# B&R Automation Studio project PickAndPlace (part 2)

#### Variables.var - Local variables
```iecst
(*FB for creating a frame and reading the status of the TrackingPath*)
VAR
	MC_ReadActualPosition_Mot1 : MC_ReadActualPosition; (*FB to read the actual axis position. Used to latch the conveyor position into each created tracking frame*)
END_VAR
(*Taking Pictures*)
VAR
	CameraPV : Camera_Type := (0); (*Camera interface struct: parameters, status, input and raw detection output from the vision function*)
	ViBaseAxisBasedAcquisition_Fb : ViBaseAxisBasedAcquisition := (0); (*FB for axis-based image acquisition. Triggers images along the axis at a fixed spatial period*)
END_VAR
(*StateMachine*)
VAR CONSTANT
	MaxObjectDetectable : USINT := 8; (*Max number of objects to manage per acquisition/filtering cycle and to size arrays accordingly*)
END_VAR
VAR
	VisionState : VisionState_Enum; (*High-level vision state machine: handles readiness, acquisition, processing, frame creation, and reset*)
	Pos_mm : ARRAY[0..MaxObjectDetectable] OF Coordinate_mm_Type := [9((0))]; (*Object positions in millimeters after pixel->mm affine transform; indexed like filtered detections*)
	i : USINT := 0; (*Generic loop index for iterating detections and buffers*)
END_VAR
(**)
VAR
	UserDataSingleItemObjectRed : TrackingFrameUserDataType := (PositionType:=SingleItemPosition,SingleItemPositionData:=(PositionFilled:=TRUE,ObjectType:=Red,SyncPosUp:=(Pos:=(Z:=10+OBJECT_HEIGHT_mm)))); (*User data attached to frames for RED objects: single-item handling with Z sync offset.*)
	UserDataSingleItemObjectBlack : TrackingFrameUserDataType := (PositionType:=SingleItemPosition,SingleItemPositionData:=(PositionFilled:=TRUE,ObjectType:=Black,SyncPosUp:=(Pos:=(Z:=10+OBJECT_HEIGHT_mm)))); (*User data attached to frames for BLACK objects: single-item handling with Z sync offset.*)
	McTrkFramesDetectedObjArray : ARRAY[0..MaxObjectDetectable] OF McTrkFrmCreateParType := [9((0))]; (*Staging buffer of frames to create for all newly detected objects in the current cycle.*)
	MC_BR_DetectedObjFramesCreat : MC_BR_TrackingFramesCreate := (0); (*FB to push the staged frames (position/orientation/attributes) to the tracking path*)
END_VAR
(**)
VAR
	LastAcquisitionCount : USINT := 0; (*Memo of the last completed acquisition index to detect new images/events from the camera*)
END_VAR
(*GetTrackingPathData*)
VAR
	TrackingPathGetFramesPos_Fb : MC_BR_TrackingPathGetFrames := (0); (*FB to read existing frames on the tracking path, used to avoid creating near-duplicate frames.*)
	FramesInfo : ARRAY[0..15] OF McTrkFrmInfoType := [16((0))]; (*Buffer holding info about up to 16 existing frames fetched from the tracking path*)
	TrackingPathGetFramesPar : McTrkPathGetFrmParType := (0); (*Parameter block for the TrackingPathGetFrames FB: modes, count, and data address*)
	j : UINT := 0; (*Secondary loop index (e.g., for distance checks against existing frames or filtered objects)*)
	RedObjectFound : BOOL := FALSE; (*Flag for the current RED candidate: TRUE if not near any stored BLACK detection (valid), FALSE if too close and discarded as duplicate.*)
	CreateNewFrame : BOOL := FALSE; (*Flag deciding whether the current detection results in a new frame after distance and overlap checks*)
	Distance_px : LREAL := 0.0; (*Euclidean distance in pixels between the current suspected RED candidate and each stored BLACK detection.*)
	Distance : LREAL := 0.0; (*Computed Euclidean distance used for de-duplication/overlap checks (units: mm in frame creation step; pixels in filtering step)*)
END_VAR
VAR CONSTANT
	OBJECT_MIN_DIST : USINT := 35; (*Minimum allowed distance (mm) between a new frame and existing frames to avoid duplicates on the tracking path.*)
END_VAR
VAR
	NumbersNewFrame : USINT := 0; (*Number of frames prepared in the current cycle to be created on the tracking path. Results after the filtering*)
	CameraOutputFiltered : VF_Output_Type := (0); (*Filtered detection list combining BLACK-first and then RED objects while avoiding overlaps/doubles*)
END_VAR
(**)
VAR
	NumBlackObj : USINT := 0; (*Number of black objects detected by the camera. This value is also used when filtering red objects, since the detection models may overlap (one detects all objects, the other only black). The variable is updated at each acquisition with the current count of detected black objects.*)
END_VAR
```

#### Init.st - Init camera and getframe FB 
```iecst
ACTION CameraInitialization:
	CameraPV.Param.GainLevel := 1;
	CameraPV.Param.SetFocus := 56000;
	CameraPV.Param.ExposureTime := 2000;
	CameraPV.Param.FlashColor := 99;
	CameraPV.Param.FlashSegment := 15;
	CameraPV.Input.EnableVF := TRUE;
	CameraPV.Input.NumSearchMax := MaxObjectDetectable;
END_ACTION

ACTION GetFramesInfoInitialization:
	TrackingPathGetFramesPos_Fb.TrackingPath := ADR(gTrackingPath_1);
	TrackingPathGetFramesPar.GetMode := mcTRKPATH_GET_MOD_ALL_FRAMES;
	TrackingPathGetFramesPar.InfoMode := mcTRKPATH_INFO_MOD_ALL;
	TrackingPathGetFramesPar.NumberOfFrames := 16;
	TrackingPathGetFramesPar.DataAddress := ADR(FramesInfo);
	TrackingPathGetFramesPos_Fb.Parameters := TrackingPathGetFramesPar;
END_ACTION
```

#### FilteringOutput.st - Builds a filtered list of detections from the raw camera output
```iecst
(**
 * Derive position and color of the physical objects from the detected shapes:
 *
 * - model=2 detects only black objects, model=1 detects black and red objects
 * - Builds a filtered list of detections from the raw camera output. It first collects all BLACK objects (Model=2) into the filtered buffer.
 * - Then it evaluates each RED candidate (Model=1) and checks its Euclidean distance in pixel space against every stored BLACK object.
 * - If a RED is closer than the configured threshold (e.g., ˜100 px when using a 10000 threshold after SQRT), it is rejected to prevent counting the same physical object twice.
 * - Valid RED detections (those not overlapping a BLACK) are appended after the BLACK entries, resulting in an ordered list: BLACK first, then non-overlapping RED.
*)
ACTION CameraOutputFiltering:

	CameraOutputFiltered.NumObjFound := 0;

	FOR i := 0 TO (CameraPV.Output.NumObjFound-1)   DO

		IF CameraPV.Output.Obj[i].Model = 2 THEN
			CameraOutputFiltered.Obj[CameraOutputFiltered.NumObjFound] := CameraPV.Output.Obj[i];
			CameraOutputFiltered.NumObjFound := CameraOutputFiltered.NumObjFound + 1;
		END_IF

	END_FOR

	NumBlackObj := CameraOutputFiltered.NumObjFound;

	FOR i := 0 TO (CameraPV.Output.NumObjFound-1)   DO

		IF CameraPV.Output.Obj[i].Model = 1 THEN
			RedObjectFound := TRUE;

			IF NumBlackObj > 0 THEN

				FOR j := 0 TO NumBlackObj-1 DO
					Distance_px := SQRT(
					brmpow(LREAL_TO_REAL(CameraPV.Output.Obj[i].Pos.X - CameraOutputFiltered.Obj[j].Pos.X ), 2) +
					brmpow(LREAL_TO_REAL(CameraPV.Output.Obj[i].Pos.Y - CameraOutputFiltered.Obj[j].Pos.Y ), 2)
					);

					IF Distance_px < 10000 THEN
						RedObjectFound := FALSE;
						EXIT;
					END_IF

				END_FOR

			END_IF

			IF RedObjectFound THEN
				CameraOutputFiltered.Obj[CameraOutputFiltered.NumObjFound] := CameraPV.Output.Obj[i];
				CameraOutputFiltered.NumObjFound := CameraOutputFiltered.NumObjFound + 1;
			END_IF

		END_IF
	END_FOR

END_ACTION
```

### Program Logical/Tasks/BufferInit (IEC) - Creation of initial objects on buffer register (PLC application task)

#### Variables.var
```iecst
VAR CONSTANT
	CONV_SLOTS_MAX_IND : USINT := CONV_SLOTS-1;
	GRID : USINT := 50; (*distance between object in the register among the y direction*)
	CONV_SLOTS : USINT := 32; (*how many object can the register contain*)
	ROWS : USINT := 4; (*rows of the register*)
END_VAR
VAR
	j : USINT := 0;
	MC_BR_TrackingFrameCreate_0 : MC_BR_TrackingFramesCreate;
	TrkFrmsToCreateOnBufferRegister : ARRAY[0..CONV_SLOTS_MAX_IND] OF McTrkFrmCreateParType;
END_VAR
(*Insert your comment here.*)
VAR
	UserDataSingleItemObjectRed : TrackingFrameUserDataType := (SubFramesVisu:=[(Attribute:=RedObjectPhysicallyPresent),4(0)],PositionType:=SingleItemPosition,SingleItemPositionData:=(PositionFilled:=TRUE,ObjectType:=Red,SyncPosUp:=(Pos:=(Z:=10+OBJECT_HEIGHT_mm))));
	UserDataSingleItemObjectBlack : TrackingFrameUserDataType := (SubFramesVisu:=[(Attribute:=BlackObjectPhysicallyPresent),4(0)],PositionType:=SingleItemPosition,SingleItemPositionData:=(PositionFilled:=TRUE,ObjectType:=Black,SyncPosUp:=(Pos:=(Z:=10+OBJECT_HEIGHT_mm))));
END_VAR
```

#### Main.st
```iecst
(**
 * Buffer Initialization
 *
 * This program initializes the buffer register with a predefined grid of objects.
 * Creates tracking frames for objects positioned in a structured layout that will serve
 * as the initial inventory for the pick-and-place operations.
 *
 * Grid Layout: Objects are arranged in a rectangular grid pattern with alternating colors
 * Pattern: Red and black objects alternate (even indices = red, odd indices = black)
 * Purpose: Provides initial objects for Robot 1 to pick from buffer and place on conveyor 2
 *)

PROGRAM _INIT

	// Creation of initial objects on buffer register

	FOR j := 0 TO CONV_SLOTS_MAX_IND DO
		// X-position: Column calculation - distributes objects across columns
		TrkFrmsToCreateOnBufferRegister[j].Translation.X := GRID / 2 + GRID * (j / ROWS);
		// Y-position: Row calculation - cycles through rows (0, 1, 2, ... ROWS-1)
		TrkFrmsToCreateOnBufferRegister[j].Translation.Y := GRID / 2 + GRID * (j MOD ROWS);
		// Z-position: Object height above the buffer surface
		TrkFrmsToCreateOnBufferRegister[j].Translation.Z := OBJECT_HEIGHT_mm;

		// Alternate between red and black objects for demonstration/testing purposes
		IF (j MOD 2 = 0) THEN
			// Even indices: Red objects
			TrkFrmsToCreateOnBufferRegister[j].Attribute := HasRedObj;
			TrkFrmsToCreateOnBufferRegister[j].UserDataAddress := ADR(UserDataSingleItemObjectRed);
		ELSE
			// Odd indices: Black objects
			TrkFrmsToCreateOnBufferRegister[j].Attribute := HasBlackObj;
			TrkFrmsToCreateOnBufferRegister[j].UserDataAddress := ADR(UserDataSingleItemObjectBlack);
		END_IF;
	END_FOR;

	MC_BR_TrackingFrameCreate_0.Parameters.DataAddress := ADR(TrkFrmsToCreateOnBufferRegister);
	MC_BR_TrackingFrameCreate_0.Parameters.NumberOfFrames := CONV_SLOTS;
	MC_BR_TrackingFrameCreate_0.TrackingPath := ADR(gTrackingPath_3);

	MC_BR_TrackingFrameCreate_0.Execute := TRUE;
	MC_BR_TrackingFrameCreate_0();

END_PROGRAM

PROGRAM _EXIT
	MC_BR_TrackingFrameCreate_0();
	MC_BR_TrackingFrameCreate_0.Execute := FALSE;
END_PROGRAM
```

### Package Logical/UserPartitionData - On transfer this folder will be copied to PLC's user partition

### Package Logical/UserPartitionData/RobotMotionPrgDir - Robot programs (Motion Structured Text)

### PnpRobot1.st - Robot 1 - Single object picker (MotionST program)
```iecst
#include 'HelperFunctions.st'
#pragma LOAD 'SharedConstants.var'

(**
 * This program controls robot 1 movements and the object selection.
 * Robot 1 has a gripper for pick single products only.
 * Robot 1 has the following pick-and-place jobs to execute:
 *		1. Pick red products from conveyor belt 1 and place them to conveyor belt 2
 *		2. Pick black products from conveyor belt 1 and place them to conveyor belt 2
 *		3. Pick red products from conveyor belt 1 and place them to buffer between the conveyor belts
 *		4. Pick black products from conveyor belt 1 and place them to buffer between the conveyor belts
 *		5. Pick red products from buffer and place them to conveyor belt 2
 *		6. Pick black products from buffer and place them to conveyor belt 2
 *
 * Priority of the jobs
 *	1. Try to find an available pick-and-place sequence for job 1 or 2:
 *		1.1 Try to find a container that that will go out of workspace next and has empty positions (HasEmptyPosForRedObj|HasEmptyPosForBlackObj)
 * 			1.1.1 Try to find a pick position that can fill this container (black or red object) (HasRedObj||HasBlackObj)
 * 	2. Alternatively when no full pick-and-place sequence is available, search for a pick position only, to initiate job 3 or job 4:
 * 		2.1 First search for pick position on conveyor belt 1, when no place position is available on conveyor 2
 * 			2.1.1 Place the object to buffer (job 3 or job 4)
 * 			2.1.2 Go to waiting position with the object in the hand and wait for place positions on conveyor 2 (job 1 or job 2)
 * 	3. If no pick position available execute job 5 or job 6:
 * 		3.1 Search for products on buffer and place them on conveyor 2 (job 5 or job 6)
 *)

VAR CONSTANT
	ParkPosWithoutObject	: McPointType 	:= (Pos:=(X:=200, Y:=200, Z:= -800));
	ParkPosWithObject		: McPointType 	:= (Pos:=(X:=-200, Y:=-200, Z:= -800));
END_VAR

VAR {AT 'Mechanics'}
	MotionProgramRob1 : RobotMotionProgramType;
END_VAR

// Robot 1 helper functions

(**
 * Selects the optimal pick and place positions for the next robot operation based on priority logic.
 * Implements the job priority system: first tries complete pick-place sequences (jobs 1-2),
 * then pick-only operations to buffer (jobs 3-4), finally buffer-to-conveyor operations (jobs 5-6).
 * Automatically updates TrackingFrame UserData and Attributes for selected positions.
 *
 * @param MotionProgram: RobotMotionProgramType - IN_OUT: Motion program structure to update with selected positions
 *)
FUNCTION SelectPickPlacePositionAndSetPnpSequenceData : BOOL
	VAR_IN_OUT
		MotionProgram : RobotMotionProgramType;
	END_VAR
	VAR
		i : UINT;
	END_VAR

	// PRIORITY 1: Try to find complete pick-place sequence (jobs 1-2)
	// First, look for containers on conveyor 2 that need filling
	TrackingFrameSelectorSetAttributeMasks('Rob1_Place_Conveyor2', 0, TrackingFrameAttributeBits#HasEmptyPosForRedObj OR TrackingFrameAttributeBits#HasEmptyPosForBlackObj, 0);
	IF TrackingFrameSelect(MotionProgram.Place.TrackingFrame.ID, 'Rob1_Place_Conveyor2') THEN
		TrackingFrameGetUserData(ADR(MotionProgram.Place.TrackingFrame.UserData),
								SIZEOF(MotionProgram.Place.TrackingFrame.UserData),
								MotionProgram.Place.TrackingFrame.ID);
		// Container found on conveyor 2 - now find matching objects on conveyor 1
		FOR i := 0 TO MAX_CONTAINER_POS_INDEX DO
			IF NOT MotionProgram.Place.TrackingFrame.UserData.ContainerPositionData.ContainedPositions[i].PositionFilled THEN
				IF MotionProgram.Place.TrackingFrame.UserData.ContainerPositionData.ContainedPositions[i].ObjectType = ObjectTypeEnum#Red THEN
					// Look for red object on conveyor 1 to fill red container slot

					TrackingFrameSelectorSetAttributeMasks('Rob1_Pick_Conveyor1', 0, TrackingFrameAttributeBits#HasRedObj, 0);
					IF TrackingFrameSelect(MotionProgram.Pick.TrackingFrame.ID, 'Rob1_Pick_Conveyor1') THEN
						TrackingFrameGetUserData(ADR(MotionProgram.Pick.TrackingFrame.UserData),
												SIZEOF(MotionProgram.Pick.TrackingFrame.UserData),
												MotionProgram.Pick.TrackingFrame.ID);
						SetPickPositionBasedOnUserData(MotionProgram, TRUE, FALSE, FALSE);
						SetPlacePositionBasedOnUserData(MotionProgram, TRUE, FALSE, FALSE);
						// Complete pick-place sequence found for red object (job 1)
						EXIT; // exit for loop
					END_IF

				ELSE // Container slot expects black object
					// Look for black object on conveyor 1 to fill black container slot

					TrackingFrameSelectorSetAttributeMasks('Rob1_Pick_Conveyor1', 0, TrackingFrameAttributeBits#HasBlackObj, 0);
					IF TrackingFrameSelect(MotionProgram.Pick.TrackingFrame.ID, 'Rob1_Pick_Conveyor1') THEN
						TrackingFrameGetUserData(ADR(MotionProgram.Pick.TrackingFrame.UserData),
												SIZEOF(MotionProgram.Pick.TrackingFrame.UserData),
												MotionProgram.Pick.TrackingFrame.ID);
						SetPickPositionBasedOnUserData(MotionProgram, FALSE, TRUE, FALSE);
						SetPlacePositionBasedOnUserData(MotionProgram, FALSE, TRUE, FALSE);
						// Complete pick-place sequence found for black object (job 2)
						EXIT; // exit for loop
					END_IF
				END_IF
			END_IF
		END_FOR;

	END_IF

	// PRIORITY 2: No complete sequence found - try pick-only operations (jobs 3-4)
	IF MotionProgram.Pick.PositionSelected=FALSE THEN

		// No pick/place combination found -> Search only for pick position
		TrackingFrameSelectorSetAttributeMasks('Rob1_Pick_Conveyor1', 0, TrackingFrameAttributeBits#HasRedObj OR TrackingFrameAttributeBits#HasBlackObj, 0);
		IF TrackingFrameSelect(MotionProgram.Pick.TrackingFrame.ID, 'Rob1_Pick_Conveyor1') THEN
			TrackingFrameGetUserData(ADR(MotionProgram.Pick.TrackingFrame.UserData),
									SIZEOF(MotionProgram.Pick.TrackingFrame.UserData),
									MotionProgram.Pick.TrackingFrame.ID);
			SetPickPositionBasedOnUserData(MotionProgram, TRUE, TRUE, FALSE);
			// Robot will PickObject
		ELSE
			TrackingFrameSelectorSetAttributeMasks('Rob1_Place_Conveyor2', 0, TrackingFrameAttributeBits#HasEmptyPosForRedObj OR TrackingFrameAttributeBits#HasEmptyPosForBlackObj, 0);
			IF TrackingFrameSelect(MotionProgram.Place.TrackingFrame.ID, 'Rob1_Place_Conveyor2')  THEN
				TrackingFrameGetUserData(ADR(MotionProgram.Place.TrackingFrame.UserData),
										SIZEOF(MotionProgram.Place.TrackingFrame.UserData),
										MotionProgram.Place.TrackingFrame.ID);
				// Expected here: Container object is present on the container placeholder position
				FOR i := 0 TO MAX_CONTAINER_POS_INDEX DO
					IF NOT MotionProgram.Place.TrackingFrame.UserData.ContainerPositionData.ContainedPositions[i].PositionFilled THEN
						IF MotionProgram.Place.TrackingFrame.UserData.ContainerPositionData.ContainedPositions[i].ObjectType = ObjectTypeEnum#Red THEN

							TrackingFrameSelectorSetAttributeMasks('Rob1_PickPlace_Buffer', 0, TrackingFrameAttributeBits#HasRedObj, 0);
							IF TrackingFrameSelect(MotionProgram.Pick.TrackingFrame.ID, 'Rob1_PickPlace_Buffer') THEN
								TrackingFrameGetUserData(ADR(MotionProgram.Pick.TrackingFrame.UserData),
														SIZEOF(MotionProgram.Pick.TrackingFrame.UserData),
														MotionProgram.Pick.TrackingFrame.ID);
								SetPickPositionBasedOnUserData(MotionProgram, TRUE, FALSE, FALSE);
								SetPlacePositionBasedOnUserData(MotionProgram, TRUE, FALSE, FALSE);
								// Robot will PickObject
								EXIT; // exit for loop
							END_IF

						ELSE // TrackingFrameUserData_Place.ContainerPositionData.ContainedPositions[i].ObjectType = ObjectTypeEnum#Black
							TrackingFrameSelectorSetAttributeMasks('Rob1_PickPlace_Buffer', 0, TrackingFrameAttributeBits#HasBlackObj, 0);
							IF TrackingFrameSelect(MotionProgram.Pick.TrackingFrame.ID, 'Rob1_PickPlace_Buffer') THEN
								TrackingFrameGetUserData(ADR(MotionProgram.Pick.TrackingFrame.UserData),
														SIZEOF(MotionProgram.Pick.TrackingFrame.UserData),
														MotionProgram.Pick.TrackingFrame.ID);
								SetPickPositionBasedOnUserData(MotionProgram, FALSE, TRUE, FALSE);
								SetPlacePositionBasedOnUserData(MotionProgram, FALSE, TRUE, FALSE);
								// Robot will PickObject
								EXIT; // exit for loop
							END_IF
						END_IF
					END_IF
				END_FOR;
			END_IF
		END_IF

		// No positions selected
	END_IF
END_FUNCTION

(**
 * Selects an appropriate place position for an object that was already picked but has no place destination.
 * This function handles scenarios where the robot picked an object but couldn't immediately find a place position.
 * Prioritizes conveyor 2 containers, falls back to buffer positions if needed.
 *
 * @param MotionProgram: RobotMotionProgramType - IN_OUT: Motion program with picked object data
 *)
FUNCTION  SelectPlacePositionAndSetPlacementData : BOOL
	VAR_IN_OUT
		MotionProgram : RobotMotionProgramType;
	END_VAR
	VAR
		i : UINT;
	END_VAR

	// 1. Check type of already picked object and select place position accordingly
	IF MotionProgram.PickedObject.Type = ObjectTypeEnum#Red THEN
		TrackingFrameSelectorSetAttributeMasks('Rob1_Place_Conveyor2', 0, TrackingFrameAttributeBits#HasEmptyPosForRedObj, 0);
	ELSE // MotionProgram.PickedObject.Type = ObjectTypeEnum#Black
		TrackingFrameSelectorSetAttributeMasks('Rob1_Place_Conveyor2', 0, TrackingFrameAttributeBits#HasEmptyPosForBlackObj, 0);
	END_IF

	IF TrackingFrameSelect(MotionProgram.Place.TrackingFrame.ID, 'Rob1_Place_Conveyor2') THEN
		TrackingFrameGetUserData(ADR(MotionProgram.Place.TrackingFrame.UserData),
								SIZEOF(MotionProgram.Place.TrackingFrame.UserData),
								MotionProgram.Place.TrackingFrame.ID);
		SetPlacePositionBasedOnUserData(MotionProgram,
										MotionProgram.PickedObject.Type=ObjectTypeEnum#Red,
										MotionProgram.PickedObject.Type=ObjectTypeEnum#Black);
	ELSE
		FOR i := 0 TO MAX_CONTAINER_POS_INDEX DO
			IF MotionProgram.PickedObject.Type = ObjectTypeEnum#Red THEN
				TrackingFrameSelectorSetAttributeMasks('Rob1_PickPlace_Buffer', 0, TrackingFrameAttributeBits#HasEmptyPosForRedObj, 0);
				IF TrackingFrameSelect(MotionProgram.Place.TrackingFrame.ID, 'Rob1_PickPlace_Buffer') THEN
					TrackingFrameGetUserData(ADR(MotionProgram.Place.TrackingFrame.UserData),
											SIZEOF(MotionProgram.Place.TrackingFrame.UserData),
											MotionProgram.Place.TrackingFrame.ID);
					SetPlacePositionBasedOnUserData(MotionProgram, TRUE, FALSE);
					// Robot will PickObject
					EXIT; // exit for loop
				END_IF

			ELSE // MotionProgram.PickedObject.Type = ObjectTypeEnum#Black
				TrackingFrameSelectorSetAttributeMasks('Rob1_PickPlace_Buffer', 0, TrackingFrameAttributeBits#HasEmptyPosForBlackObj, 0);
				IF TrackingFrameSelect(MotionProgram.Place.TrackingFrame.ID, 'Rob1_PickPlace_Buffer') THEN
					TrackingFrameGetUserData(ADR(MotionProgram.Place.TrackingFrame.UserData),
											SIZEOF(MotionProgram.Place.TrackingFrame.UserData),
											MotionProgram.Place.TrackingFrame.ID);
					SetPlacePositionBasedOnUserData(MotionProgram, FALSE, TRUE);
					// Robot will PickObject
					EXIT;
				END_IF

			END_IF
		END_FOR;
	END_IF

END_FUNCTION

(**
 * Main selection function for pick and place positions when robot has no object.
 * Calls the detailed selection logic and determines the next robot state based on results.
 * Handles parking behavior when no suitable positions are found.
 *
 * @param MotionProgram: RobotMotionProgramType - IN_OUT: Motion program structure to update
 * @param FromPlacePos: BOOL - TRUE if coming from place position, FALSE if from waiting position
 *)
FUNCTION SelectPickPlacePosition : BOOL
	VAR_IN_OUT
		MotionProgram : RobotMotionProgramType;
	END_VAR
	VAR_INPUT
		FromPlacePos : BOOL; // TRUE: coming from place position, FALSE: coming from waiting position
	END_VAR

	MotionProgram.Pick.PositionSelected := FALSE;
	MotionProgram.Place.PositionSelected := FALSE;
	SelectPickPlacePositionAndSetPnpSequenceData(MotionProgram);
	IF MotionProgram.Pick.PositionSelected AND MotionProgram.Place.PositionSelected THEN
		MotionProgram.State := RobotStateEnum#PickObject;
	ELSIF MotionProgram.Pick.PositionSelected THEN
		MotionProgram.State := RobotStateEnum#PickObject;
	ELSE
		IF FromPlacePos THEN
			TrackStopR(MachineFrame, ParkPosWithoutObject, 50, 50);
			WaitEndMove();
		END_IF
		MotionProgram.State := RobotStateEnum#ParkWithNoObject;
	END_IF
END_FUNCTION

(**
 * Selects a place position for an object already held by the robot.
 * Used when robot picked an object but couldn't immediately find a place destination.
 * Handles parking behavior with object when no place position is available.
 *
 * @param MotionProgram: RobotMotionProgramType - IN_OUT: Motion program with picked object data
 * @param FromPickPos: BOOL - TRUE if coming from pick position, FALSE if from waiting position
 *)
FUNCTION SelectPlacePosition : BOOL
	VAR_IN_OUT
		MotionProgram : RobotMotionProgramType;
	END_VAR
	VAR_INPUT
		FromPickPos : BOOL; // TRUE: coming from pick position, FALSE: coming from waiting position
	END_VAR
	MotionProgram.Place.PositionSelected := FALSE;
	SelectPlacePositionAndSetPlacementData(MotionProgram);
	IF MotionProgram.Place.PositionSelected THEN
		MotionProgram.State:=RobotStateEnum#PlaceObject;
	ELSE
		IF FromPickPos THEN
			TrackStopR(MachineFrame, ParkPosWithObject, 50, 50);
			WaitEndMove();
		END_IF
		MotionProgram.State := RobotStateEnum#ParkWithGrippedObject;
	END_IF

END_FUNCTION

(**
 * Updates the products in the gripper to be shown in Scene Viewer
 *)
FUNCTION UpdateGripperContent : BOOL
	VAR_IN_OUT
		MotionProgram : RobotMotionProgramType;
	END_VAR
	VAR_INPUT
		Pick : BOOL; // TRUE: Pick operation, FALSE: Place operation
	END_VAR
	IF Pick THEN
		MotionProgram.GripperContent.RedObjectInGripper[0] := MotionProgram.PickedObject.Type = ObjectTypeEnum#Red;
		MotionProgram.GripperContent.BlackObjectInGripper[0] := MotionProgram.PickedObject.Type = ObjectTypeEnum#Black;
	ELSE
		MotionProgram.GripperContent.RedObjectInGripper[0] := FALSE;
		MotionProgram.GripperContent.BlackObjectInGripper[0] := FALSE;
	END_IF
END_FUNCTION

// Robot 1 Main Motion Program - State Machine Implementation

PROGRAM _MAIN

	MotionProgramRob1.State := RobotStateEnum#Start;

	REPEAT
		CASE MotionProgramRob1.State OF

			RobotStateEnum#Start:
				// Initialize robot to park position without object
				MoveLR(ParkPosWithoutObject);
				WaitALAP();
				MotionProgramRob1.State := RobotStateEnum#ParkWithNoObject;

			RobotStateEnum#PickObject:
				// Execute pick operation
				TrackObjectR(MotionProgramRob1.Pick.TrackingFrame.ID, MotionProgramRob1.Pick.SynchPosUp, 50, 50);
				DO_PATH_SYNCH
					MotionProgramRob1.CloseGripper := TRUE;	 // To increase throughput (reduce required WaitTime), also signaling feature could be used for activating the vaccuum
				END_PATH_SYNCH
				MoveLR(MotionProgramRob1.Pick.SynchPosDown);
				DO_PATH_SYNCH
					UpdateGripperContent(MotionProgramRob1, TRUE);
				END_PATH_SYNCH
				WaitTime(0.2);
				MoveLR(MotionProgramRob1.Pick.SynchPosUp);
				IF MotionProgramRob1.Place.PositionSelected THEN
					MotionProgramRob1.State := RobotStateEnum#PlaceObject;
				ELSE
					WaitALAP();
					SelectPlacePosition(MotionProgramRob1, TRUE);
				END_IF

			RobotStateEnum#PlaceObject:
				// Execute place operation
				TrackObjectR(MotionProgramRob1.Place.TrackingFrame.ID, MotionProgramRob1.Place.SynchPosUp, 50, 50);
				MoveLR(MotionProgramRob1.Place.SynchPosDown);
				DO_PATH_SYNCH
					MotionProgramRob1.CloseGripper := FALSE;	 // To increase throughput (reduce required WaitTime), also signaling feature could be used for deactivating the vaccuum
					UpdateGripperContent(MotionProgramRob1, FALSE);
				END_PATH_SYNCH
				WaitTime(0.1);
				MoveLR(MotionProgramRob1.Place.SynchPosUp);
				WaitALAP();
				// Look for next pick-place sequence after successful placement
				SelectPickPlacePosition(MotionProgramRob1, TRUE);

			RobotStateEnum#ParkWithNoObject:
				// Robot is parked without object - continuously search for work
				SelectPickPlacePosition(MotionProgramRob1, FALSE);

			RobotStateEnum#ParkWithGrippedObject:
				// Robot has object but no place position - search for place destination
				SelectPlacePosition(MotionProgramRob1, FALSE);

		END_CASE
	UNTIL FALSE END_REPEAT;

END_PROGRAM
```

### PnpRobot2.st - Robot 2 - Container picker (MotionST program)
```iecst
#include 'HelperFunctions.st'
#pragma LOAD 'SharedConstants.var'

(**
 * This program controls robot 2 movements and object selection.
 * Robot 2 has a gripper designed for picking entire containers (4 objects at once).
 * Robot 2 has a single pick-and-place job to execute:
 *		Pick complete containers that have been filled by robot 1 from conveyor belt 2
 *		and place them on conveyor belt 1.
 *
 * Operation: Robot 2 waits for containers on conveyor 2 that contain objects (filled by Robot 1),
 * then transfers these complete containers to conveyor 1.
 *)

VAR CONSTANT
	ParkPosWithoutObject      : McPointType := (Pos:=(X:=-200, Y:=-200, Z:= -800));
	ParkPosWithObject      : McPointType := (Pos:=(X:=200, Y:=200, Z:= -800));
END_VAR
VAR {AT 'Mechanics'}
	MotionProgramRob2 : RobotMotionProgramType;
END_VAR

// Robot 2 helper functions

(**
 * Selects a filled container on conveyor 2 for picking operation.
 * Searches for containers that contain objects (filled by Robot 1) and are ready for transfer.
 * Automatically updates TrackingFrame UserData and Attributes for the selected position.
 *
 * @param MotionProgram: RobotMotionProgramType - IN_OUT: Motion program structure to update with pick position
 *)
FUNCTION SelectPickPositionAndSetPickData : BOOL
	VAR_IN_OUT
		MotionProgram : RobotMotionProgramType;
	END_VAR
	VAR
		i : UINT;
	END_VAR

	// Search for containers on conveyor 2 that contain objects (red or black)
	TrackingFrameSelectorSetAttributeMasks('Rob2_Pick_Conveyor2', 0, TrackingFrameAttributeBits#HasRedObj OR TrackingFrameAttributeBits#HasBlackObj, 0);

	IF TrackingFrameSelect(MotionProgram.Pick.TrackingFrame.ID, 'Rob2_Pick_Conveyor2') THEN
		TrackingFrameGetUserData(ADR(MotionProgram.Pick.TrackingFrame.UserData),
								SIZEOF(MotionProgram.Pick.TrackingFrame.UserData),
								MotionProgram.Pick.TrackingFrame.ID);
		SetPickPositionBasedOnUserData(MotionProgram, FALSE, FALSE, TRUE);
		// Container selected for pickup
	END_IF
END_FUNCTION

(**
 * Selects an empty container position on conveyor 1 for placing the picked container.
 * Searches for available container placeholder positions on the destination conveyor.
 * Automatically updates TrackingFrame UserData and Attributes for the selected position.
 *
 * @param MotionProgram: RobotMotionProgramType - IN_OUT: Motion program structure to update with place position
 *)
FUNCTION  SelectPlacePositionAndSetPlacementData : BOOL
	VAR_IN_OUT
		MotionProgram : RobotMotionProgramType;
	END_VAR
	VAR
		i : UINT;
	END_VAR

	// Search for empty container positions on conveyor 1
	TrackingFrameSelectorSetAttributeMasks('Rob2_Place_Conveyor1', 0, TrackingFrameAttributeBits#HasEmptyPosForContainer, 0);
	IF TrackingFrameSelect(MotionProgram.Place.TrackingFrame.ID, 'Rob2_Place_Conveyor1') THEN
		TrackingFrameGetUserData(ADR(MotionProgram.Place.TrackingFrame.UserData),
								SIZEOF(MotionProgram.Place.TrackingFrame.UserData),
								MotionProgram.Place.TrackingFrame.ID);
		SetPlacePositionBasedOnUserData(MotionProgram, FALSE, FALSE, TRUE);
	END_IF
END_FUNCTION

(**
 * Main selection function for pick positions when robot has no container.
 * Calls the detailed pick selection logic and determines the next robot state based on results.
 * Handles parking behavior when no suitable containers are available for pickup.
 *
 * @param MotionProgram: RobotMotionProgramType - IN_OUT: Motion program structure to update
 * @param FromPlacePos: BOOL - TRUE if coming from place position, FALSE if from waiting position
 *)
FUNCTION SelectPickPosition : BOOL
	VAR_IN_OUT
		MotionProgram : RobotMotionProgramType;
	END_VAR
	VAR_INPUT
		FromPlacePos : BOOL; // TRUE: coming from place position, FALSE: coming from waiting position
	END_VAR
	MotionProgram.Pick.PositionSelected := FALSE;
	SelectPickPositionAndSetPickData(MotionProgram);
	IF MotionProgram.Pick.PositionSelected THEN
		MotionProgram.State := RobotStateEnum#PickObject;
	ELSE
		IF FromPlacePos THEN
			TrackStopR(MachineFrame, ParkPosWithoutObject, 50, 50);
			WaitEndMove();
		END_IF
		MotionProgram.State := RobotStateEnum#ParkWithNoObject;
	END_IF

END_FUNCTION

(**
 * Selects a place position for a container already held by the robot.
 * Used when robot picked a container but couldn't immediately find a place destination.
 * Handles parking behavior with container when no place position is available.
 *
 * @param MotionProgram: RobotMotionProgramType - IN_OUT: Motion program with picked container data
 * @param FromPickPos: BOOL - TRUE if coming from pick position, FALSE if from waiting position
 *)
FUNCTION SelectPlacePosition : BOOL
	VAR_IN_OUT
		MotionProgram : RobotMotionProgramType;
	END_VAR
	VAR_INPUT
		FromPickPos : BOOL; // TRUE: coming from pick position, FALSE: coming from waiting position
	END_VAR
	MotionProgram.Place.PositionSelected := FALSE;
	SelectPlacePositionAndSetPlacementData(MotionProgram);
	IF MotionProgram.Place.PositionSelected THEN
		MotionProgram.State:=RobotStateEnum#PlaceObject;
	ELSE
		IF FromPickPos THEN
			TrackStopR(MachineFrame, ParkPosWithObject, 50, 50);
			WaitEndMove();
		END_IF
		MotionProgram.State:=RobotStateEnum#ParkWithGrippedObject;
	END_IF
END_FUNCTION

(**
 *  * Updates the products in the gripper to be shown in Scene Viewer
 *)
FUNCTION UpdateGripperContent : BOOL
	VAR_IN_OUT
		MotionProgram : RobotMotionProgramType;
	END_VAR
	VAR_INPUT
		Pick : BOOL; // TRUE: Pick operation, FALSE: Place operation
	END_VAR
	IF Pick THEN
		MotionProgram.GripperContent.RedObjectInGripper[0] := MotionProgram.Pick.TrackingFrame.UserData.ContainerPositionData.ContainedPositions[0].PositionFilled AND MotionProgram.Pick.TrackingFrame.UserData.ContainerPositionData.ContainedPositions[0].ObjectType = ObjectTypeEnum#Red;
		MotionProgram.GripperContent.RedObjectInGripper[1] := MotionProgram.Pick.TrackingFrame.UserData.ContainerPositionData.ContainedPositions[1].PositionFilled AND MotionProgram.Pick.TrackingFrame.UserData.ContainerPositionData.ContainedPositions[1].ObjectType = ObjectTypeEnum#Red;
		MotionProgram.GripperContent.RedObjectInGripper[2] := MotionProgram.Pick.TrackingFrame.UserData.ContainerPositionData.ContainedPositions[2].PositionFilled AND MotionProgram.Pick.TrackingFrame.UserData.ContainerPositionData.ContainedPositions[2].ObjectType = ObjectTypeEnum#Red;
		MotionProgram.GripperContent.RedObjectInGripper[3] := MotionProgram.Pick.TrackingFrame.UserData.ContainerPositionData.ContainedPositions[3].PositionFilled AND MotionProgram.Pick.TrackingFrame.UserData.ContainerPositionData.ContainedPositions[3].ObjectType = ObjectTypeEnum#Red;

		MotionProgram.GripperContent.BlackObjectInGripper[0] := MotionProgram.Pick.TrackingFrame.UserData.ContainerPositionData.ContainedPositions[0].PositionFilled AND MotionProgram.Pick.TrackingFrame.UserData.ContainerPositionData.ContainedPositions[0].ObjectType = ObjectTypeEnum#Black;
		MotionProgram.GripperContent.BlackObjectInGripper[1] := MotionProgram.Pick.TrackingFrame.UserData.ContainerPositionData.ContainedPositions[1].PositionFilled AND MotionProgram.Pick.TrackingFrame.UserData.ContainerPositionData.ContainedPositions[1].ObjectType = ObjectTypeEnum#Black;
		MotionProgram.GripperContent.BlackObjectInGripper[2] := MotionProgram.Pick.TrackingFrame.UserData.ContainerPositionData.ContainedPositions[2].PositionFilled AND MotionProgram.Pick.TrackingFrame.UserData.ContainerPositionData.ContainedPositions[2].ObjectType = ObjectTypeEnum#Black;
		MotionProgram.GripperContent.BlackObjectInGripper[3] := MotionProgram.Pick.TrackingFrame.UserData.ContainerPositionData.ContainedPositions[3].PositionFilled AND MotionProgram.Pick.TrackingFrame.UserData.ContainerPositionData.ContainedPositions[3].ObjectType = ObjectTypeEnum#Black;
	ELSE
		MotionProgram.GripperContent.RedObjectInGripper[0] := FALSE;
		MotionProgram.GripperContent.RedObjectInGripper[1] := FALSE;
		MotionProgram.GripperContent.RedObjectInGripper[2] := FALSE;
		MotionProgram.GripperContent.RedObjectInGripper[3] := FALSE;

		MotionProgram.GripperContent.BlackObjectInGripper[0] := FALSE;
		MotionProgram.GripperContent.BlackObjectInGripper[1] := FALSE;
		MotionProgram.GripperContent.BlackObjectInGripper[2] := FALSE;
		MotionProgram.GripperContent.BlackObjectInGripper[3] := FALSE;
	END_IF
END_FUNCTION

// Robot 2 Main Motion Program - Container Transfer State Machine

PROGRAM _MAIN

	MotionProgramRob2.State := RobotStateEnum#Start;

	REPEAT
		CASE MotionProgramRob2.State OF

			RobotStateEnum#Start:
				// Initialize robot to park position
				MoveLR(ParkPosWithoutObject);
				WaitALAP();
				MotionProgramRob2.State := RobotStateEnum#ParkWithNoObject;

			RobotStateEnum#PickObject:
				// Execute container pick operation
				TrackObjectR(MotionProgramRob2.Pick.TrackingFrame.ID, MotionProgramRob2.Pick.SynchPosUp, 50, 50);
				DO_PATH_SYNCH
					MotionProgramRob2.CloseGripper := TRUE;	 // To increase throughput (reduce required WaitTime), also signaling feature could be used for deactivating the vaccuum
				END_PATH_SYNCH
				MoveLR(MotionProgramRob2.Pick.SynchPosDown);
				DO_PATH_SYNCH
					UpdateGripperContent(MotionProgramRob2, TRUE);
				END_PATH_SYNCH
				WaitTime(0.1); // Allow time for container to settle in gripper
				MoveLR(MotionProgramRob2.Pick.SynchPosUp);
				WaitALAP();
				// Search for place position after successful container pickup
				SelectPlacePosition(MotionProgramRob2, TRUE);

			RobotStateEnum#PlaceObject:
				// Execute container place operation
				TrackObjectR(MotionProgramRob2.Place.TrackingFrame.ID, MotionProgramRob2.Place.SynchPosUp, 50, 50);
				MoveLR(MotionProgramRob2.Place.SynchPosDown);
				DO_PATH_SYNCH
					MotionProgramRob2.CloseGripper := FALSE;	 // To increase throughput (reduce required WaitTime), also signaling feature could be used for deactivating the vaccuum
					UpdateGripperContent(MotionProgramRob2, FALSE);
				END_PATH_SYNCH
				WaitTime(0.05); // Brief wait for container release
				MoveLR(MotionProgramRob2.Place.SynchPosUp);
				WaitALAP();
				// Look for next container to transfer after successful placement
				SelectPickPosition(MotionProgramRob2, TRUE);

			RobotStateEnum#ParkWithNoObject:
				// Robot is parked without container - continuously search for containers to transfer
				SelectPickPosition(MotionProgramRob2, FALSE);

			RobotStateEnum#ParkWithGrippedObject:
				// Robot has container but no place position - search for place destination
				SelectPlacePosition(MotionProgramRob2, FALSE);

		END_CASE
	UNTIL FALSE END_REPEAT;

END_PROGRAM
```

### HelperFunctions.st - Helper functions for objects selection shared by both robots (MotionST functions)
```iecst
#include 'SharedTypes.typ'
#pragma LOAD 'SharedConstants.var'

(*
 * Generates and returns an attribute value (bitmask) that represents the state of the TrackingFrame userData.
 * This function analyzes the position type and object states to create appropriate attribute flags.
 *
 * @param userData: TrackingFrameUserDataType - The user data structure containing position and object information
 * @return UDINT - Bitmask representing the current state (empty positions, object types, etc.)
 *)
FUNCTION GetAttributeBasedOnUserData : UDINT
	VAR_INPUT
		userData : TrackingFrameUserDataType;
	END_VAR
	VAR
		attribute : UDINT;
		i : UINT;
	END_VAR
	attribute := 0;
	IF userData.PositionType = TrackingFramePositionTypeEnum#SingleItemPosition THEN
		IF userData.SingleItemPositionData.PositionFilled = FALSE THEN
			IF userData.SingleItemPositionData.ObjectType = ObjectTypeEnum#Red THEN
				attribute := attribute OR TrackingFrameAttributeBits#HasEmptyPosForRedObj;
			ELSE // userData.SingleItemPositionData.ObjectType = ObjectTypeEnum#Black
				attribute := attribute OR TrackingFrameAttributeBits#HasEmptyPosForBlackObj;
			END_IF
		ELSE // userData.SingleItemPositionData.PositionFilled = TRUE
			IF userData.SingleItemPositionData.ObjectType = ObjectTypeEnum#Red THEN
				attribute := attribute OR TrackingFrameAttributeBits#HasRedObj;
			ELSE // userData.SingleItemPositionData.ObjectType = ObjectTypeEnum#Black
				attribute := attribute OR TrackingFrameAttributeBits#HasBlackObj;
			END_IF
		END_IF
	ELSIF userData.PositionType = TrackingFramePositionTypeEnum#ContainerPosition THEN
		IF userData.ContainerPositionData.PositionFilled = FALSE THEN
			attribute := attribute OR TrackingFrameAttributeBits#HasEmptyPosForContainer;
		ELSE //userData.ContainerPositionData.PositionFilled = TRUE
			FOR i := 0 TO MAX_CONTAINER_POS_INDEX DO
				IF userData.ContainerPositionData.ContainedPositions[i].PositionFilled THEN
					IF userData.ContainerPositionData.ContainedPositions[i].ObjectType = ObjectTypeEnum#Red THEN
						attribute := attribute OR TrackingFrameAttributeBits#HasRedObj;
					ELSE // userData.ContainerPositionData.ContainedPositions[i].ObjectType = ObjectTypeEnum#Black
						attribute := attribute OR TrackingFrameAttributeBits#HasBlackObj;
					END_IF
				ELSE // userData.ContainerPositionData.ContainedPositions[i].PositionFilled = FALSE
					IF userData.ContainerPositionData.ContainedPositions[i].ObjectType = ObjectTypeEnum#Red THEN
						attribute := attribute OR TrackingFrameAttributeBits#HasEmptyPosForRedObj;
					ELSE // userData.ContainerPositionData.ContainedPositions[i].ObjectType = ObjectTypeEnum#Black
						attribute := attribute OR TrackingFrameAttributeBits#HasEmptyPosForBlackObj;
					END_IF
				END_IF
			END_FOR;
		END_IF
	END_IF
	GetAttributeBasedOnUserData := attribute;
END_FUNCTION

(*
 * Generates an attribute value (bitmask) and writes it directly to the specified TrackingFrame.
 * This is a convenience function that combines GetAttributeBasedOnUserData with TrackingFrameSetAttribute.
 *
 * @param trackingFrameId: McTrkFrmIdentType - The ID of the tracking frame to update
 * @param userData: TrackingFrameUserDataType - The user data to analyze for attribute generation
 * @return UDINT - The generated attribute bitmask that was written to the tracking frame
 *)
FUNCTION SetAttributeBasedOnUserData : UDINT
	VAR_INPUT
		trackingFrameId : McTrkFrmIdentType;
		userData : TrackingFrameUserDataType;
	END_VAR
	VAR
		attribute : UDINT;
	END_VAR
	attribute := GetAttributeBasedOnUserData(userData);
	TrackingFrameSetAttribute(trackingFrameId, attribute);
	SetAttributeBasedOnUserData := attribute;
END_FUNCTION

(*
 * Configures the pick operation in the MotionProgram based on selected TrackingFrame userData.
 * Updates synchronization positions, object type information, and marks the position as empty after picking.
 *
 * @param MotionProgram: RobotMotionProgramType - IN_OUT: Motion program structure to update
 * @param objectTypeRed: BOOL - TRUE if red objects should be considered for picking
 * @param objectTypeBlack: BOOL - TRUE if black objects should be considered for picking
 * @param objectTypeContainer: BOOL - TRUE to pick entire container, FALSE to pick individual contained item
 * @return BOOL - Success status of the operation
 *)
FUNCTION SetPickPositionBasedOnUserData : BOOL
	VAR_IN_OUT
		MotionProgram : RobotMotionProgramType;
	END_VAR
	VAR_INPUT
		objectTypeRed : BOOL;
		objectTypeBlack : BOOL;
		objectTypeContainer : BOOL; // TRUE the entire container will be picked, FALSE only a contained item will be picked
	END_VAR
	VAR
		i : UINT;
	END_VAR
	IF MotionProgram.Pick.TrackingFrame.UserData.PositionType = TrackingFramePositionTypeEnum#SingleItemPosition THEN
		MotionProgram.Pick.SynchPosUp := MotionProgram.Pick.TrackingFrame.UserData.SingleItemPositionData.SyncPosUp;
		MotionProgram.Pick.SynchPosDown := MotionProgram.Pick.TrackingFrame.UserData.SingleItemPositionData.SyncPosDown;
		MotionProgram.PickedObject.Type := MotionProgram.Pick.TrackingFrame.UserData.SingleItemPositionData.ObjectType;
		MotionProgram.PickedObject.ContainerIndex := 0; // No container index for single item position
		MotionProgram.Pick.TrackingFrame.UserData.SingleItemPositionData.PositionFilled := FALSE;
		MotionProgram.Pick.TrackingFrame.UserData.SubFramesVisu[0].Attribute := MotionProgram.Pick.TrackingFrame.UserData.SubFramesVisu[0].Attribute OR TrackingFrameAttributeBits#ProductSelectedForOperation;
	ELSE // MotionProgram.Pick.TrackingFrame.UserData.PositionType = TrackingFramePositionTypeEnum#ContainerPosition
		IF objectTypeContainer THEN // Entire container will be picked
			MotionProgram.Pick.SynchPosUp := MotionProgram.Pick.TrackingFrame.UserData.ContainerPositionData.SyncPosUp;
			MotionProgram.Pick.SynchPosDown := MotionProgram.Pick.TrackingFrame.UserData.ContainerPositionData.SyncPosDown;
			MotionProgram.Pick.TrackingFrame.UserData.ContainerPositionData.PositionFilled := FALSE;
			MotionProgram.Pick.TrackingFrame.UserData.SubFramesVisu[0].Attribute := MotionProgram.Pick.TrackingFrame.UserData.SubFramesVisu[0].Attribute OR TrackingFrameAttributeBits#ContainerSelectedForOperation;
		ELSE // Only a contained item will be picked
			// Search through container positions to find the requested object type
			FOR i := 0 TO MAX_CONTAINER_POS_INDEX DO
				IF MotionProgram.Pick.TrackingFrame.UserData.ContainerPositionData.ContainedPositions[i].PositionFilled THEN
					IF objectTypeRed AND MotionProgram.Pick.TrackingFrame.UserData.ContainerPositionData.ContainedPositions[i].ObjectType = ObjectTypeEnum#Red THEN
						MotionProgram.Pick.SynchPosUp := MotionProgram.Pick.TrackingFrame.UserData.ContainerPositionData.ContainedPositions[i].SyncPosUp;
						MotionProgram.Pick.SynchPosDown := MotionProgram.Pick.TrackingFrame.UserData.ContainerPositionData.ContainedPositions[i].SyncPosDown;
						MotionProgram.PickedObject.Type := MotionProgram.Pick.TrackingFrame.UserData.ContainerPositionData.ContainedPositions[i].ObjectType;
						MotionProgram.PickedObject.ContainerIndex := i;
						MotionProgram.Pick.TrackingFrame.UserData.ContainerPositionData.ContainedPositions[i].PositionFilled := FALSE;
						MotionProgram.Pick.TrackingFrame.UserData.SubFramesVisu[i+1].Attribute := MotionProgram.Pick.TrackingFrame.UserData.SubFramesVisu[i+1].Attribute OR TrackingFrameAttributeBits#ProductSelectedForOperation;
						EXIT; // exit for loop
					ELSIF objectTypeBlack AND MotionProgram.Pick.TrackingFrame.UserData.ContainerPositionData.ContainedPositions[i].ObjectType = ObjectTypeEnum#Black THEN
						MotionProgram.Pick.SynchPosUp := MotionProgram.Pick.TrackingFrame.UserData.ContainerPositionData.ContainedPositions[i].SyncPosUp;
						MotionProgram.Pick.SynchPosDown := MotionProgram.Pick.TrackingFrame.UserData.ContainerPositionData.ContainedPositions[i].SyncPosDown;
						MotionProgram.PickedObject.Type := MotionProgram.Pick.TrackingFrame.UserData.ContainerPositionData.ContainedPositions[i].ObjectType;
						MotionProgram.PickedObject.ContainerIndex := i;
						MotionProgram.Pick.TrackingFrame.UserData.ContainerPositionData.ContainedPositions[i].PositionFilled := FALSE;
						MotionProgram.Pick.TrackingFrame.UserData.SubFramesVisu[i+1].Attribute := MotionProgram.Pick.TrackingFrame.UserData.SubFramesVisu[i+1].Attribute OR TrackingFrameAttributeBits#ProductSelectedForOperation;
						EXIT; // exit for loop
					END_IF
				END_IF
			END_FOR;

		END_IF
	END_IF
	MotionProgram.Pick.PositionSelected := TRUE;
	TrackingFrameSetUserData(ADR(MotionProgram.Pick.TrackingFrame.UserData),
							SIZEOF(MotionProgram.Pick.TrackingFrame.UserData),
							MotionProgram.Pick.TrackingFrame.ID);
	MotionProgram.Pick.TrackingFrame.Attribute := SetAttributeBasedOnUserData(MotionProgram.Pick.TrackingFrame.ID, MotionProgram.Pick.TrackingFrame.UserData);
END_FUNCTION

(*
 * Configures the place operation in the MotionProgram based on selected TrackingFrame userData.
 * Updates synchronization positions, transfers object data from pick to place position, and marks position as filled.
 *
 * @param MotionProgram: RobotMotionProgramType - IN_OUT: Motion program structure to update
 * @param objectTypeRed: BOOL - TRUE if red objects should be considered for placement
 * @param objectTypeBlack: BOOL - TRUE if black objects should be considered for placement
 * @param objectTypeContainer: BOOL - TRUE to place entire container, FALSE to place individual item in container
 * @return BOOL - Success status of the operation
 *)
FUNCTION SetPlacePositionBasedOnUserData : BOOL
	VAR_IN_OUT
		MotionProgram : RobotMotionProgramType;
	END_VAR
	VAR_INPUT
		objectTypeRed : BOOL;
		objectTypeBlack : BOOL;
		objectTypeContainer : BOOL; // TRUE the entire container will be picked, FALSE only a contained item will be picked
	END_VAR
	VAR
		i : UINT;
	END_VAR
	IF MotionProgram.Place.TrackingFrame.UserData.PositionType = TrackingFramePositionTypeEnum#SingleItemPosition THEN
		MotionProgram.Place.SynchPosUp := MotionProgram.Place.TrackingFrame.UserData.SingleItemPositionData.SyncPosUp;
		MotionProgram.Place.SynchPosDown := MotionProgram.Place.TrackingFrame.UserData.SingleItemPositionData.SyncPosDown;
		// Transfer product identification from pick to place position for traceability
		MotionProgram.Place.TrackingFrame.UserData.SingleItemPositionData.ProductID := MotionProgram.Pick.TrackingFrame.UserData.SingleItemPositionData.ProductID;
		MotionProgram.Place.TrackingFrame.UserData.SingleItemPositionData.PositionFilled := TRUE;
		MotionProgram.Place.TrackingFrame.UserData.SubFramesVisu[0].Attribute := MotionProgram.Place.TrackingFrame.UserData.SubFramesVisu[0].Attribute OR TrackingFrameAttributeBits#ProductSelectedForOperation;
	ELSE // MotionProgram.Place.TrackingFrame.UserData.PositionType = TrackingFramePositionTypeEnum#ContainerPosition
		IF objectTypeContainer THEN // Entire container will be placed
			MotionProgram.Place.SynchPosUp := MotionProgram.Place.TrackingFrame.UserData.ContainerPositionData.SyncPosUp;
			MotionProgram.Place.SynchPosDown := MotionProgram.Place.TrackingFrame.UserData.ContainerPositionData.SyncPosDown;
			MotionProgram.Place.TrackingFrame.UserData.ContainerPositionData := MotionProgram.Pick.TrackingFrame.UserData.ContainerPositionData; // Copy container data from pick to place position
			MotionProgram.Place.TrackingFrame.UserData.ContainerPositionData.PositionFilled := TRUE;
			MotionProgram.Place.TrackingFrame.UserData.SubFramesVisu[0].Attribute := MotionProgram.Place.TrackingFrame.UserData.SubFramesVisu[0].Attribute OR TrackingFrameAttributeBits#ContainerSelectedForOperation;
		ELSE // Will be placed in a contained position only
			// Search for position with object present
			FOR i := 0 TO MAX_CONTAINER_POS_INDEX DO
				IF NOT MotionProgram.Place.TrackingFrame.UserData.ContainerPositionData.ContainedPositions[i].PositionFilled THEN
					IF objectTypeRed AND MotionProgram.Place.TrackingFrame.UserData.ContainerPositionData.ContainedPositions[i].ObjectType = ObjectTypeEnum#Red THEN
						MotionProgram.Place.SynchPosUp := MotionProgram.Place.TrackingFrame.UserData.ContainerPositionData.ContainedPositions[i].SyncPosUp;
						MotionProgram.Place.SynchPosDown := MotionProgram.Place.TrackingFrame.UserData.ContainerPositionData.ContainedPositions[i].SyncPosDown;
						MotionProgram.Place.TrackingFrame.UserData.ContainerPositionData.ContainedPositions[i].ProductID :=
							MotionProgram.Pick.TrackingFrame.UserData.ContainerPositionData.ContainedPositions[MotionProgram.PickedObject.ContainerIndex].ProductID;
						MotionProgram.Place.TrackingFrame.UserData.ContainerPositionData.ContainedPositions[i].PositionFilled := TRUE;
						MotionProgram.Place.TrackingFrame.UserData.SubFramesVisu[i+1].Attribute := MotionProgram.Place.TrackingFrame.UserData.SubFramesVisu[i+1].Attribute OR TrackingFrameAttributeBits#ProductSelectedForOperation;
						EXIT; // exit for loop
					ELSIF objectTypeBlack AND MotionProgram.Place.TrackingFrame.UserData.ContainerPositionData.ContainedPositions[i].ObjectType = ObjectTypeEnum#Black THEN
						MotionProgram.Place.SynchPosUp := MotionProgram.Place.TrackingFrame.UserData.ContainerPositionData.ContainedPositions[i].SyncPosUp;
						MotionProgram.Place.SynchPosDown := MotionProgram.Place.TrackingFrame.UserData.ContainerPositionData.ContainedPositions[i].SyncPosDown;
						MotionProgram.Place.TrackingFrame.UserData.ContainerPositionData.ContainedPositions[i].ProductID :=
							MotionProgram.Pick.TrackingFrame.UserData.ContainerPositionData.ContainedPositions[MotionProgram.PickedObject.ContainerIndex].ProductID;
						MotionProgram.Place.TrackingFrame.UserData.ContainerPositionData.ContainedPositions[i].PositionFilled := TRUE;
						MotionProgram.Place.TrackingFrame.UserData.SubFramesVisu[i+1].Attribute := MotionProgram.Place.TrackingFrame.UserData.SubFramesVisu[i+1].Attribute OR TrackingFrameAttributeBits#ProductSelectedForOperation;
						EXIT; // exit for loop
					END_IF
				END_IF
			END_FOR;
		END_IF
	END_IF
	MotionProgram.Place.PositionSelected := TRUE;
	TrackingFrameSetUserData(ADR(MotionProgram.Place.TrackingFrame.UserData),
							SIZEOF(MotionProgram.Place.TrackingFrame.UserData),
							MotionProgram.Place.TrackingFrame.ID);
	MotionProgram.Place.TrackingFrame.Attribute := SetAttributeBasedOnUserData(MotionProgram.Place.TrackingFrame.ID, MotionProgram.Place.TrackingFrame.UserData);
END_FUNCTION

(**
 * Updates the products on conveyor shown in Scene Viewer
 *)
FUNCTION UpdateConveyorContent : BOOL
	VAR_IN_OUT
		TrkFrmId : McTrkFrmIdentType;
		TrkFrmUserData : TrackingFrameUserDataType;
	END_VAR
	VAR
		i : UINT;
	END_VAR

	TrackingFrameGetUserData(ADR(TrkFrmUserData), SIZEOF(TrkFrmUserData), TrkFrmId);

	IF TrkFrmUserData.PositionType = TrackingFramePositionTypeEnum#SingleItemPosition THEN

		TrkFrmUserData.SubFramesVisu[0].Pos := TrkFrmUserData.SingleItemPositionData.SyncPosDown.Pos;
		TrkFrmUserData.SubFramesVisu[0].Orient := TrkFrmUserData.SingleItemPositionData.SyncPosDown.Orient;
		IF TrkFrmUserData.SingleItemPositionData.PositionFilled THEN
			IF TrkFrmUserData.SingleItemPositionData.ObjectType = ObjectTypeEnum#Red THEN
				TrkFrmUserData.SubFramesVisu[0].Attribute := TrackingFrameAttributeBits#RedObjectPhysicallyPresent;
			ELSE
				TrkFrmUserData.SubFramesVisu[0].Attribute := TrackingFrameAttributeBits#BlackObjectPhysicallyPresent;
			END_IF
		ELSE
			TrkFrmUserData.SubFramesVisu[0].Attribute := 0;
		END_IF

	ELSE // MotionProgram.Pick.TrackingFrame.UserData.PositionType = TrackingFramePositionTypeEnum#ContainerPosition

		TrkFrmUserData.SubFramesVisu[0].Pos := TrkFrmUserData.ContainerPositionData.SyncPosDown.Pos;
		TrkFrmUserData.SubFramesVisu[0].Orient := TrkFrmUserData.ContainerPositionData.SyncPosDown.Orient;

		IF TrkFrmUserData.ContainerPositionData.PositionFilled THEN
			TrkFrmUserData.SubFramesVisu[0].Attribute := 0; // Overwrite object selection marker
			FOR i := 0 TO MAX_CONTAINER_POS_INDEX DO
				//offset i+1: 1st sub frame is the container itself
				TrkFrmUserData.SubFramesVisu[i+1].Pos := TrkFrmUserData.ContainerPositionData.ContainedPositions[i].SyncPosDown.Pos;
				TrkFrmUserData.SubFramesVisu[i+1].Orient := TrkFrmUserData.ContainerPositionData.ContainedPositions[i].SyncPosDown.Orient;
				IF TrkFrmUserData.ContainerPositionData.ContainedPositions[i].PositionFilled THEN
					IF TrkFrmUserData.ContainerPositionData.ContainedPositions[i].ObjectType = ObjectTypeEnum#Red THEN
						TrkFrmUserData.SubFramesVisu[i+1].Attribute := TrackingFrameAttributeBits#RedObjectPhysicallyPresent;
					ELSE
						TrkFrmUserData.SubFramesVisu[i+1].Attribute := TrackingFrameAttributeBits#BlackObjectPhysicallyPresent;
					END_IF
				ELSE
					TrkFrmUserData.SubFramesVisu[i+1].Attribute := 0;
				END_IF
			END_FOR;
		ELSE
			TrkFrmUserData.SubFramesVisu[0].Attribute := 0;
			TrkFrmUserData.SubFramesVisu[1].Attribute := 0;
			TrkFrmUserData.SubFramesVisu[2].Attribute := 0;
			TrkFrmUserData.SubFramesVisu[3].Attribute := 0;
			TrkFrmUserData.SubFramesVisu[4].Attribute := 0;
		END_IF

	END_IF

	TrackingFrameSetUserData(ADR(TrkFrmUserData), SIZEOF(TrkFrmUserData), TrkFrmId);

END_FUNCTION
```

### SharedConstants.var - Shared constants that are used in motion program and PLC application task
```iecst
VAR CONSTANT
	MAX_CONTAINER_POS_INDEX : UINT := 3; (*'Number of single item positions in a container' minus 1*)
END_VAR
```

### SharedTypes.typ - Shared data types that are used in motion program and PLC application task
```iecst
(*TrackingFrame user data*)

TYPE
	TrackingFrameUserDataType : 	STRUCT
		SubFramesVisu : ARRAY[0..4]OF McTrkFrmSubFrmType;
		PositionType : TrackingFramePositionTypeEnum;
		SingleItemPositionData : SingleItemPositionDataType;
		ContainerPositionData : ContainerPositionDataType;
	END_STRUCT;
	TrackingFramePositionTypeEnum :
		(
		SingleItemPosition := 0,
		ContainerPosition := 1
		);
	SingleItemPositionDataType : 	STRUCT
		PositionFilled : BOOL;
		ObjectType : ObjectTypeEnum;
		ProductID : UDINT; (*Optional: ID of product*)
		SyncPosUp : McPointType;
		SyncPosDown : McPointType;
	END_STRUCT;
	ContainerPositionDataType : 	STRUCT
		PositionFilled : BOOL;
		ContainedPositions : ARRAY[0..MAX_CONTAINER_POS_INDEX]OF SingleItemPositionDataType;
		ContainerID : UDINT; (*Optional: ID of container*)
		SyncPosUp : McPointType;
		SyncPosDown : McPointType;
	END_STRUCT;
	ObjectTypeEnum :
		(
		Red := 0,
		Black := 1
		);
	RobotStateEnum :
		(
		Start := 0,
		PickObject := 1,
		PlaceObject := 2,
		ParkWithNoObject := 3,
		ParkWithGrippedObject := 4
		);
END_TYPE

(*Motion Program*)

TYPE
	RobotMotionProgramType : 	STRUCT
		Pick : RobotMotionPickPlaceType;
		Place : RobotMotionPickPlaceType;
		PickedObject : PickedObjectType;
		State : RobotStateEnum;
		CloseGripper : BOOL;
		GripperContent : GripperContentType;
		CleaningMachine : BOOL;
	END_STRUCT;
	RobotMotionPickPlaceType : 	STRUCT
		PositionSelected : BOOL;
		TrackingFrame : RobotMotionTrkFrmType;
		SynchPosUp : McPointType;
		SynchPosDown : McPointType;
	END_STRUCT;
	RobotMotionTrkFrmType : 	STRUCT
		ID : McTrkFrmIdentType;
		UserData : TrackingFrameUserDataType;
		Attribute : UDINT;
	END_STRUCT;
	PickedObjectType : 	STRUCT
		Type : ObjectTypeEnum;
		ContainerIndex : UINT; (*Use for pick/place positions in a container only*)
	END_STRUCT;
	GripperContentType : 	STRUCT
		RedObjectInGripper : ARRAY[0..3]OF BOOL;
		BlackObjectInGripper : ARRAY[0..3]OF BOOL;
	END_STRUCT;
END_TYPE

(*TrackingFrame and SubFrame attribute: Bit code*)

TYPE
	TrackingFrameAttributeBits :
		(
		HasEmptyPosForRedObj := 2#00000000000000000000000000000001, (*Object selection synchronous state of a TrackingFrame (used for TrackingFrame selection)*)
		HasEmptyPosForBlackObj := 2#00000000000000000000000000000010, (*Object selection synchronous state of a TrackingFrame (used for TrackingFrame selection)*)
		HasRedObj := 2#00000000000000000000000000000100, (*Object selection synchronous state of a TrackingFrame (used for TrackingFrame selection)*)
		HasBlackObj := 2#00000000000000000000000000001000, (*Object selection synchronous state of a TrackingFrame (used for TrackingFrame selection)*)
		HasEmptyPosForContainer := 2#00000000000000000000000000010000, (*Object selection synchronous state of a TrackingFrame (used for TrackingFrame selection)*)
		RedObjectPhysicallyPresent := 2#00000000000000000000000000100000, (*Movement synchronous state of a SubFrame (used for 3D visu)*)
		BlackObjectPhysicallyPresent := 2#00000000000000000000000001000000, (*Movement synchronous state of a SubFrame  (used for 3D visu)*)
		ProductSelectedForOperation := 2#00000000000000000000000010000000, (*Object selection synchronous state of a SubFrame  (used for 3D visu)*)
		ContainerSelectedForOperation := 2#00000000000000000000000100000000 (*Object selection synchronous state of a SubFrame  (used for 3D visu)*)
		);
END_TYPE
```
